{attribute 'qualified_only'}
VAR_GLOBAL
	// Test Motors
	M1 : DUT_MotionStage;
	M2 : DUT_MotionStage;
	
	// Test Encoders
	stMasterEnc : ST_RenishawAbsEnc;
	stSlaveEnc : ST_RenishawAbsEnc;
END_VAR

(* stored: Version 1.1.0.1, ProductVersion 3.1.4022.18
   GVL GVL_GantryInterlockStopsMotion: Id {c06e4a3c-aeb8-43ef-8fac-1752f505e7e0} *)
